// TIA Portal V21 export
DATA_BLOCK "BatchTempOnOff"   // DB300
// stored: AutoNumber false, InstanceOfName FB104, InstanceOfType FB
"FB104"
   // VAR_INPUT
   //    Enable : Bool;
   //    SecPulse : Bool;
   //    AlwaysTrue : Bool;
   //    DigitalOrAnalog : Bool;
   //    InvertPIDSel : Bool;
   //    ActValue : Real;
   //    SetValue : Real;
   //    SetPoint1 : Real;
   //    SetPoint2 : Real;
   //    SetPoint3 : Real;
   //    SetPoint4 : Real;
   //    SetPoint5 : Real;
   //    SetPoint6 : Real;
   //    SetPoint7 : Real;
   //    SetPoint8 : Real;
   //    SetPoint9 : Real;
   //    SetPoint10 : Real;
   //    SetRef1 : Real;
   //    SetRef2 : Real;
   //    SetRef3 : Real;
   //    SetRef4 : Real;
   //    SetRef5 : Real;
   //    SetRef6 : Real;
   //    SetRef7 : Real;
   //    SetRef8 : Real;
   //    SetRef9 : Real;
   //    SetRef10 : Real;
   //    OnTime1 : Int;
   //    OnTime2 : Int;
   //    OnTime3 : Int;
   //    OnTime4 : Int;
   //    OnTime5 : Int;
   //    OnTime6 : Int;
   //    OnTime7 : Int;
   //    OnTime8 : Int;
   //    OnTime9 : Int;
   //    OnTime10 : Int;
   //    OffTime1 : Int;
   //    OffTime2 : Int;
   //    OffTime3 : Int;
   //    OffTime4 : Int;
   //    OffTime5 : Int;
   //    OffTime6 : Int;
   //    OffTime7 : Int;
   //    OffTime8 : Int;
   //    OffTime9 : Int;
   //    OffTime10 : Int;
   // END_VAR
   // VAR_OUTPUT
   //    Valve : Bool;
   //    SetRef : Real;
   // END_VAR
   // VAR_IN_OUT
   //    ControlValue1 : Real;
   //    ControlValue2 : Real;
   //    ControlValue3 : Real;
   //    ControlValue4 : Real;
   //    ControlValue5 : Real;
   //    ControlValue6 : Real;
   //    ControlValue7 : Real;
   //    ControlValue8 : Real;
   //    ControlValue9 : Real;
   //    ControlValue10 : Real;
   // END_VAR
   // VAR
   //    OnOffDelay { S7_SetPoint := 'True'} : "FB102";
   //    OnTime : Int;
   //    OffTime : Int;
   // END_VAR
BEGIN
END_DATA_BLOCK
